ABB RAPID module: Robtargets.mod

MODULE Robtargets

    !**************************************************************************
    !ROBTARGET DECLARATIONS
    !**************************************************************************
    ! HOME AND STARTING Positions.

    CONST jointtarget AbsHome:=[[0,0,0,0,90,-60],[0,9E+09,9E+09,9E+09,9E+09,9E+09]];
    CONST robtarget Home:=[[351.01,0.00,709.09],[1.0026E-05,-3.87097E-05,1,4.46769E-06],[0,0,-1,0],[9E+09,9E+09,9E+09,9E+09,9E+09,9E+09]];
    CONST robtarget AboveStartAPosition:=[[68.84,70.35,87.16],[0.128377,0.734299,0.632585,-0.210145],[-1,-1,-1,0],[9E+09,9E+09,9E+09,9E+09,9E+09,9E+09]];
    CONST robtarget StartPosition:=[[68.84,70.35,87.16],[0.128377,0.734299,0.632585,-0.210145],[-1,-1,-1,0],[9E+09,9E+09,9E+09,9E+09,9E+09,9E+09]];
    CONST robtarget DicePickupPos:=[[-9.63,16.11,24.81],[0.0168056,0.706657,0.706736,-0.0296041],[-1,0,-2,0],[9E+09,9E+09,9E+09,9E+09,9E+09,9E+09]];
    CONST robtarget DiceThrowPos:=[[77.33,10.92,132.18],[0.0426025,0.942934,-0.0615583,-0.324456],[-2,0,-2,0],[9E+09,9E+09,9E+09,9E+09,9E+09,9E+09]];
    CONST robtarget DiceAbovePickPos:=[[-9.63,16.10,87.18],[0.0167928,0.706652,0.706742,-0.0296007],[-1,0,-2,0],[9E+09,9E+09,9E+09,9E+09,9E+09,9E+09]];

    CONST robtarget WinnerPos:=[[200.71,534.63,135.22],[0.00124171,-0.715438,-0.698667,-0.00340603],[0,0,0,0],[9E+09,9E+09,9E+09,9E+09,9E+09,9E+09]];
    CONST robtarget WinnerAbovePos:=[[200.71,534.63,260],[0.00124171,-0.715438,-0.698667,-0.00340603],[0,0,0,0],[9E+09,9E+09,9E+09,9E+09,9E+09,9E+09]];


    CONST robtarget Player1StartPos:=[[-39.27,392.54,23.61],[0.00279119,-0.701491,-0.712559,-0.0127358],[-1,-1,-1,0],[9E+09,9E+09,9E+09,9E+09,9E+09,9E+09]];
    CONST robtarget AbovePlayer1StartPos:=[[-39.27,392.54,200],[0.00279119,-0.701491,-0.712559,-0.0127358],[-1,-1,-1,0],[9E+09,9E+09,9E+09,9E+09,9E+09,9E+09]];
    CONST robtarget Player2StartPos:=[[-40.43,297.08,24.03],[0.00278384,-0.701482,-0.712569,-0.0126879],[-1,-1,-1,0],[9E+09,9E+09,9E+09,9E+09,9E+09,9E+09]];
    CONST robtarget AbovePlayer2StartPos:=[[-40.43,297.08,200],[0.00278384,-0.701482,-0.712569,-0.0126879],[-1,-1,-1,0],[9E+09,9E+09,9E+09,9E+09,9E+09,9E+09]];

    CONST robtarget Position00:=[[63.18,74.54,88.95],[0.138777,0.819807,0.520878,-0.193242],[-1,-1,0,0],[9E+09,9E+09,9E+09,9E+09,9E+09,9E+09]];
    CONST robtarget AbovePosition00:=[[63.18,74.54,200],[0.138777,0.819807,0.520878,-0.193242],[-1,-1,0,0],[9E+09,9E+09,9E+09,9E+09,9E+09,9E+09]];

    !1 TO 9
    CONST robtarget Position1:=[[118.73,66.16,87.22],[0.138793,0.819813,0.520859,-0.193257],[-1,-1,0,0],[9E+09,9E+09,9E+09,9E+09,9E+09,9E+09]];
    CONST robtarget AbovePosition1:=[[118.73,66.16,200],[0.138793,0.819813,0.520859,-0.193257],[-1,-1,0,0],[9E+09,9E+09,9E+09,9E+09,9E+09,9E+09]];

    CONST robtarget Position2:=[[177.20,64.51,84.69],[0.118125,0.704224,0.692906,-0.0999847],[-1,0,-1,0],[9E+09,9E+09,9E+09,9E+09,9E+09,9E+09]];
    CONST robtarget AbovePosition2:=[[177.20,64.51,200],[0.118125,0.704224,0.692906,-0.0999847],[-1,0,-1,0],[9E+09,9E+09,9E+09,9E+09,9E+09,9E+09]];

    CONST robtarget Position3:=[[231.06,64.54,84.66],[0.118102,0.704224,0.692915,-0.0999518],[-1,0,-1,0],[9E+09,9E+09,9E+09,9E+09,9E+09,9E+09]];
    CONST robtarget AbovePosition3:=[[231.06,64.54,200],[0.118102,0.704224,0.692915,-0.0999518],[-1,0,-1,0],[9E+09,9E+09,9E+09,9E+09,9E+09,9E+09]];

    CONST robtarget Position4:=[[283.24,64.54,84.66],[0.118095,0.704232,0.692908,-0.0999451],[0,0,-1,0],[9E+09,9E+09,9E+09,9E+09,9E+09,9E+09]];
    CONST robtarget AbovePosition4:=[[283.24,64.54,200],[0.118095,0.704232,0.692908,-0.0999451],[0,0,-1,0],[9E+09,9E+09,9E+09,9E+09,9E+09,9E+09]];

    CONST robtarget Position5:=[[336.21,64.54,84.66],[0.118088,0.704236,0.692906,-0.0999428],[0,-1,0,0],[9E+09,9E+09,9E+09,9E+09,9E+09,9E+09]];
    CONST robtarget AbovePosition5:=[[336.21,64.54,200],[0.118088,0.704236,0.692906,-0.0999428],[0,-1,0,0],[9E+09,9E+09,9E+09,9E+09,9E+09,9E+09]];

    CONST robtarget Position6:=[[388.67,64.54,84.66],[0.118113,0.704241,0.692895,-0.0999498],[0,-1,0,0],[9E+09,9E+09,9E+09,9E+09,9E+09,9E+09]];
    CONST robtarget AbovePosition6:=[[388.67,64.54,200],[0.118113,0.704241,0.692895,-0.0999498],[0,-1,0,0],[9E+09,9E+09,9E+09,9E+09,9E+09,9E+09]];

    CONST robtarget Position7:=[[439.75,64.55,84.60],[0.118098,0.704233,0.692908,-0.0999314],[0,-1,0,0],[9E+09,9E+09,9E+09,9E+09,9E+09,9E+09]];
    CONST robtarget AbovePosition7:=[[439.75,64.55,200],[0.118098,0.704233,0.692908,-0.0999314],[0,-1,0,0],[9E+09,9E+09,9E+09,9E+09,9E+09,9E+09]];

    CONST robtarget Position8:=[[491.75,69.67,84.56],[0.118087,0.704245,0.692902,-0.0999056],[0,-1,0,0],[9E+09,9E+09,9E+09,9E+09,9E+09,9E+09]];
    CONST robtarget AbovePosition8:=[[491.75,69.67,200],[0.118087,0.704245,0.692902,-0.0999056],[0,-1,0,0],[9E+09,9E+09,9E+09,9E+09,9E+09,9E+09]];

    CONST robtarget Position9:=[[510.49,108.79,84.55],[0.118067,0.70425,0.692902,-0.0998953],[0,-1,0,0],[9E+09,9E+09,9E+09,9E+09,9E+09,9E+09]];
    CONST robtarget AbovePosition9:=[[510.49,108.79,200],[0.118067,0.70425,0.692902,-0.0998953],[0,-1,0,0],[9E+09,9E+09,9E+09,9E+09,9E+09,9E+09]];

    CONST robtarget Position10:=[[476.96,151.88,84.56],[0.118067,0.704252,0.6929,-0.0998956],[0,-1,0,0],[9E+09,9E+09,9E+09,9E+09,9E+09,9E+09]];
    CONST robtarget AbovePosition10:=[[476.96,151.88,200],[0.118067,0.704252,0.6929,-0.0998956],[0,-1,0,0],[9E+09,9E+09,9E+09,9E+09,9E+09,9E+09]];


    !11 TO 20

    CONST robtarget Position11:=[[423.95,153.84,84.54],[0.118026,0.704242,0.69292,-0.0998776],[0,-1,0,0],[9E+09,9E+09,9E+09,9E+09,9E+09,9E+09]];
    CONST robtarget AbovePosition11:=[[423.95,153.84,200],[0.118026,0.704242,0.69292,-0.0998776],[0,-1,0,0],[9E+09,9E+09,9E+09,9E+09,9E+09,9E+09]];

    CONST robtarget Position12:=[[370.80,153.84,84.54],[0.118025,0.704242,0.692921,-0.0998746],[0,-1,0,0],[9E+09,9E+09,9E+09,9E+09,9E+09,9E+09]];
    CONST robtarget AbovePosition12:=[[370.80,153.84,200],[0.118025,0.704242,0.692921,-0.0998746],[0,-1,0,0],[9E+09,9E+09,9E+09,9E+09,9E+09,9E+09]];

    CONST robtarget Position13:=[[316.56,153.85,84.54],[0.118018,0.704245,0.692919,-0.0998685],[0,0,0,0],[9E+09,9E+09,9E+09,9E+09,9E+09,9E+09]];
    CONST robtarget AbovePosition13:=[[316.56,153.85,200],[0.118018,0.704245,0.692919,-0.0998685],[0,0,0,0],[9E+09,9E+09,9E+09,9E+09,9E+09,9E+09]];

    CONST robtarget Position14:=[[263.55,153.85,84.54],[0.118015,0.704243,0.692922,-0.0998641],[-1,0,-1,0],[9E+09,9E+09,9E+09,9E+09,9E+09,9E+09]];
    CONST robtarget AbovePosition14:=[[263.55,153.85,200],[0.118015,0.704243,0.692922,-0.0998641],[-1,0,-1,0],[9E+09,9E+09,9E+09,9E+09,9E+09,9E+09]];

    CONST robtarget Position15:=[[211.29,153.83,84.55],[0.118027,0.704235,0.692925,-0.0998929],[-1,0,-1,0],[9E+09,9E+09,9E+09,9E+09,9E+09,9E+09]];
    CONST robtarget AbovePosition15:=[[211.29,153.83,200],[0.118027,0.704235,0.692925,-0.0998929],[-1,0,-1,0],[9E+09,9E+09,9E+09,9E+09,9E+09,9E+09]];

    CONST robtarget Position16:=[[156.95,153.83,84.55],[0.118029,0.70423,0.692928,-0.0999031],[-1,0,-1,0],[9E+09,9E+09,9E+09,9E+09,9E+09,9E+09]];
    CONST robtarget AbovePosition16:=[[156.95,153.83,200],[0.118029,0.70423,0.692928,-0.0999031],[-1,0,-1,0],[9E+09,9E+09,9E+09,9E+09,9E+09,9E+09]];

    CONST robtarget Position17:=[[106.54,161.05,84.55],[0.118023,0.704218,0.69294,-0.0999059],[-1,0,-1,0],[9E+09,9E+09,9E+09,9E+09,9E+09,9E+09]];
    CONST robtarget AbovePosition17:=[[106.54,161.05,200],[0.118023,0.704218,0.69294,-0.0999059],[-1,0,-1,0],[9E+09,9E+09,9E+09,9E+09,9E+09,9E+09]];

    CONST robtarget Position18:=[[72.88,199.41,84.55],[0.118015,0.704204,0.692958,-0.0998897],[-1,0,-1,0],[9E+09,9E+09,9E+09,9E+09,9E+09,9E+09]];
    CONST robtarget AbovePosition18:=[[72.88,199.41,200],[0.118015,0.704204,0.692958,-0.0998897],[-1,0,-1,0],[9E+09,9E+09,9E+09,9E+09,9E+09,9E+09]];

    CONST robtarget Position19:=[[90.15,247.20,83.27],[0.00101801,-0.715468,-0.698638,-0.00318642],[-1,0,-1,0],[9E+09,9E+09,9E+09,9E+09,9E+09,9E+09]];
    CONST robtarget AbovePosition19:=[[90.15,247.20,200],[0.00101801,-0.715468,-0.698638,-0.00318642],[-1,0,-1,0],[9E+09,9E+09,9E+09,9E+09,9E+09,9E+09]];

    CONST robtarget Position20:=[[144.64,258.44,83.28],[0.00102727,-0.715462,-0.698643,-0.00319756],[-1,0,-1,0],[9E+09,9E+09,9E+09,9E+09,9E+09,9E+09]];
    CONST robtarget AbovePosition20:=[[144.64,258.44,200],[0.00102727,-0.715462,-0.698643,-0.00319756],[-1,0,-1,0],[9E+09,9E+09,9E+09,9E+09,9E+09,9E+09]];


    !21 TO 30

    CONST robtarget Position21:=[[197.53,258.45,83.28],[0.00104167,-0.715455,-0.69865,-0.00321534],[-1,0,-1,0],[9E+09,9E+09,9E+09,9E+09,9E+09,9E+09]];
    CONST robtarget AbovePosition21:=[[197.53,258.45,200],[0.00104167,-0.715455,-0.69865,-0.00321534],[-1,0,-1,0],[9E+09,9E+09,9E+09,9E+09,9E+09,9E+09]];

    CONST robtarget Position22:=[[251.56,258.46,83.29],[0.00104929,-0.715452,-0.698653,-0.00322303],[-1,0,-1,0],[9E+09,9E+09,9E+09,9E+09,9E+09,9E+09]];
    CONST robtarget AbovePosition22:=[[251.56,258.46,200],[0.00104929,-0.715452,-0.698653,-0.00322303],[-1,0,-1,0],[9E+09,9E+09,9E+09,9E+09,9E+09,9E+09]];

    CONST robtarget Position23:=[[304.12,258.46,83.28],[0.00104724,-0.715454,-0.698652,-0.00322172],[0,0,0,0],[9E+09,9E+09,9E+09,9E+09,9E+09,9E+09]];
    CONST robtarget AbovePosition23:=[[304.12,258.46,200],[0.00104724,-0.715454,-0.698652,-0.00322172],[0,0,0,0],[9E+09,9E+09,9E+09,9E+09,9E+09,9E+09]];

    CONST robtarget Position24:=[[355.55,258.45,83.28],[0.00102149,-0.715468,-0.698638,-0.00320467],[0,0,0,0],[9E+09,9E+09,9E+09,9E+09,9E+09,9E+09]];
    CONST robtarget AbovePosition24:=[[355.55,258.45,200],[0.00102149,-0.715468,-0.698638,-0.00320467],[0,0,0,0],[9E+09,9E+09,9E+09,9E+09,9E+09,9E+09]];

    CONST robtarget Position25:=[[409.67,258.45,83.28],[0.00101934,-0.715458,-0.698648,-0.0032026],[0,0,0,0],[9E+09,9E+09,9E+09,9E+09,9E+09,9E+09]];
    CONST robtarget AbovePosition25:=[[409.67,258.45,200],[0.00101934,-0.715458,-0.698648,-0.0032026],[0,0,0,0],[9E+09,9E+09,9E+09,9E+09,9E+09,9E+09]];

    CONST robtarget Position26:=[[464.38,260.32,83.27],[0.00103049,-0.715445,-0.698661,-0.00320834],[0,0,0,0],[9E+09,9E+09,9E+09,9E+09,9E+09,9E+09]];
    CONST robtarget AbovePosition26:=[[464.38,260.32,200],[0.00103049,-0.715445,-0.698661,-0.00320834],[0,0,0,0],[9E+09,9E+09,9E+09,9E+09,9E+09,9E+09]];

    CONST robtarget Position27:=[[494.41,301.60,83.28],[0.00104603,-0.715438,-0.698668,-0.00321548],[0,0,0,0],[9E+09,9E+09,9E+09,9E+09,9E+09,9E+09]];
    CONST robtarget AbovePosition27:=[[494.41,301.60,200],[0.00104603,-0.715438,-0.698668,-0.00321548],[0,0,0,0],[9E+09,9E+09,9E+09,9E+09,9E+09,9E+09]];

    CONST robtarget Position28:=[[481.35,349.43,83.26],[0.00107789,-0.715427,-0.698679,-0.00321957],[0,0,0,0],[9E+09,9E+09,9E+09,9E+09,9E+09,9E+09]];
    CONST robtarget AbovePosition28:=[[481.35,349.43,200],[0.00107789,-0.715427,-0.698679,-0.00321957],[0,0,0,0],[9E+09,9E+09,9E+09,9E+09,9E+09,9E+09]];

    CONST robtarget Position29:=[[428.33,351.84,83.26],[0.00109179,-0.715424,-0.698682,-0.00322696],[0,0,0,0],[9E+09,9E+09,9E+09,9E+09,9E+09,9E+09]];
    CONST robtarget AbovePosition29:=[[428.33,351.84,200],[0.00109179,-0.715424,-0.698682,-0.00322696],[0,0,0,0],[9E+09,9E+09,9E+09,9E+09,9E+09,9E+09]];

    CONST robtarget Position30:=[[375.36,351.85,83.26],[0.00110089,-0.715426,-0.69868,-0.00323293],[0,0,0,0],[9E+09,9E+09,9E+09,9E+09,9E+09,9E+09]];
    CONST robtarget AbovePosition30:=[[375.36,351.85,200],[0.00110089,-0.715426,-0.69868,-0.00323293],[0,0,0,0],[9E+09,9E+09,9E+09,9E+09,9E+09,9E+09]];


    !31 TO 40
    CONST robtarget Position31:=[[322.93,352.08,83.25],[0.00115336,-0.715442,-0.698663,-0.00327321],[0,-1,0,0],[9E+09,9E+09,9E+09,9E+09,9E+09,9E+09]];
    CONST robtarget AbovePosition31:=[[322.93,352.08,200],[0.00115336,-0.715442,-0.698663,-0.00327321],[0,-1,0,0],[9E+09,9E+09,9E+09,9E+09,9E+09,9E+09]];

    CONST robtarget Position32:=[[269.71,352.09,83.24],[0.00116463,-0.715448,-0.698657,-0.00328896],[-1,-1,-1,0],[9E+09,9E+09,9E+09,9E+09,9E+09,9E+09]];
    CONST robtarget AbovePosition32:=[[269.71,352.09,200],[0.00116463,-0.715448,-0.698657,-0.00328896],[-1,-1,-1,0],[9E+09,9E+09,9E+09,9E+09,9E+09,9E+09]];

    CONST robtarget Position33:=[[218.15,352.10,83.24],[0.00116707,-0.71544,-0.698665,-0.00328863],[-1,-1,-1,0],[9E+09,9E+09,9E+09,9E+09,9E+09,9E+09]];
    CONST robtarget AbovePosition33:=[[218.15,352.10,200],[0.00116707,-0.71544,-0.698665,-0.00328863],[-1,-1,-1,0],[9E+09,9E+09,9E+09,9E+09,9E+09,9E+09]];

    CONST robtarget Position34:=[[164.48,352.12,83.23],[0.00117983,-0.715427,-0.698678,-0.00331468],[-1,-1,-1,0],[9E+09,9E+09,9E+09,9E+09,9E+09,9E+09]];
    CONST robtarget AbovePosition34:=[[164.48,352.12,200],[0.00117983,-0.715427,-0.698678,-0.00331468],[-1,-1,-1,0],[9E+09,9E+09,9E+09,9E+09,9E+09,9E+09]];

    CONST robtarget Position35:=[[110.09,358.92,83.22],[0.00119315,-0.715427,-0.698679,-0.00334963],[-1,-1,-1,0],[9E+09,9E+09,9E+09,9E+09,9E+09,9E+09]];
    CONST robtarget AbovePosition35:=[[110.09,358.92,200],[0.00119315,-0.715427,-0.698679,-0.00334963],[-1,-1,-1,0],[9E+09,9E+09,9E+09,9E+09,9E+09,9E+09]];

    CONST robtarget Position36:=[[60.69,378.82,83.22],[0.00119013,-0.715425,-0.698681,-0.00333409],[-1,-1,-1,0],[9E+09,9E+09,9E+09,9E+09,9E+09,9E+09]];
    CONST robtarget AbovePosition36:=[[60.69,378.82,200],[0.00119013,-0.715425,-0.698681,-0.00333409],[-1,-1,-1,0],[9E+09,9E+09,9E+09,9E+09,9E+09,9E+09]];

    CONST robtarget Position37:=[[48.55,422.87,83.23],[0.00119175,-0.71543,-0.698675,-0.00333562],[-1,-1,-1,0],[9E+09,9E+09,9E+09,9E+09,9E+09,9E+09]];
    CONST robtarget AbovePosition37:=[[48.55,422.87,200],[0.00119175,-0.71543,-0.698675,-0.00333562],[-1,-1,-1,0],[9E+09,9E+09,9E+09,9E+09,9E+09,9E+09]];

    CONST robtarget Position38:=[[85.32,456.96,83.23],[0.00119527,-0.715427,-0.698679,-0.00335135],[-1,-1,-1,0],[9E+09,9E+09,9E+09,9E+09,9E+09,9E+09]];
    CONST robtarget AbovePosition38:=[[85.32,456.96,200],[0.00119527,-0.715427,-0.698679,-0.00335135],[-1,-1,-1,0],[9E+09,9E+09,9E+09,9E+09,9E+09,9E+09]];

    CONST robtarget Position39:=[[138.35,457.61,83.23],[0.00120429,-0.715433,-0.698672,-0.00338569],[-1,-1,-1,0],[9E+09,9E+09,9E+09,9E+09,9E+09,9E+09]];
    CONST robtarget AbovePosition39:=[[138.35,457.61,200],[0.00120429,-0.715433,-0.698672,-0.00338569],[-1,-1,-1,0],[9E+09,9E+09,9E+09,9E+09,9E+09,9E+09]];

    CONST robtarget Position40:=[[191.56,457.62,83.23],[0.00121366,-0.715427,-0.698678,-0.00340316],[-1,-1,-1,0],[9E+09,9E+09,9E+09,9E+09,9E+09,9E+09]];
    CONST robtarget AbovePosition40:=[[191.56,457.62,200],[0.00121366,-0.715427,-0.698678,-0.00340316],[-1,-1,-1,0],[9E+09,9E+09,9E+09,9E+09,9E+09,9E+09]];


    !41 TO 50
    CONST robtarget Position41:=[[245.02,457.62,83.23],[0.00121799,-0.715424,-0.698681,-0.00341009],[-1,-1,-1,0],[9E+09,9E+09,9E+09,9E+09,9E+09,9E+09]];
    CONST robtarget AbovePosition41:=[[245.02,457.62,200],[0.00121799,-0.715424,-0.698681,-0.00341009],[-1,-1,-1,0],[9E+09,9E+09,9E+09,9E+09,9E+09,9E+09]];

    CONST robtarget Position42:=[[297.02,457.62,83.22],[0.00121059,-0.715423,-0.698683,-0.00340594],[0,0,0,0],[9E+09,9E+09,9E+09,9E+09,9E+09,9E+09]];
    CONST robtarget AbovePosition42:=[[297.02,457.62,200],[0.00121059,-0.715423,-0.698683,-0.00340594],[0,0,0,0],[9E+09,9E+09,9E+09,9E+09,9E+09,9E+09]];

    CONST robtarget Position43:=[[350.67,457.62,83.22],[0.00120303,-0.715424,-0.698681,-0.00340147],[0,0,0,0],[9E+09,9E+09,9E+09,9E+09,9E+09,9E+09]];
    CONST robtarget AbovePosition43:=[[350.67,457.62,200],[0.00120303,-0.715424,-0.698681,-0.00340147],[0,0,0,0],[9E+09,9E+09,9E+09,9E+09,9E+09,9E+09]];

    CONST robtarget Position44:=[[405.00,457.61,83.22],[0.00118815,-0.71543,-0.698675,-0.0033961],[0,0,0,0],[9E+09,9E+09,9E+09,9E+09,9E+09,9E+09]];
    CONST robtarget AbovePosition44:=[[405.00,457.61,200],[0.00118815,-0.71543,-0.698675,-0.0033961],[0,0,0,0],[9E+09,9E+09,9E+09,9E+09,9E+09,9E+09]];

    CONST robtarget Position45:=[[455.85,457.60,83.22],[0.00114772,-0.715425,-0.69868,-0.00338543],[0,0,0,0],[9E+09,9E+09,9E+09,9E+09,9E+09,9E+09]];
    CONST robtarget AbovePosition45:=[[455.85,457.60,200],[0.00114772,-0.715425,-0.69868,-0.00338543],[0,0,0,0],[9E+09,9E+09,9E+09,9E+09,9E+09,9E+09]];

    CONST robtarget Position46:=[[498.76,483.63,83.22],[0.0011547,-0.715421,-0.698685,-0.0033882],[0,0,0,0],[9E+09,9E+09,9E+09,9E+09,9E+09,9E+09]];
    CONST robtarget AbovePosition46:=[[498.76,483.63,200],[0.0011547,-0.715421,-0.698685,-0.0033882],[0,0,0,0],[9E+09,9E+09,9E+09,9E+09,9E+09,9E+09]];

    CONST robtarget Position47:=[[492.42,526.12,83.22],[0.0011983,-0.715428,-0.698677,-0.00339119],[0,0,0,0],[9E+09,9E+09,9E+09,9E+09,9E+09,9E+09]];
    CONST robtarget AbovePosition47:=[[492.42,526.12,200],[0.0011983,-0.715428,-0.698677,-0.00339119],[0,0,0,0],[9E+09,9E+09,9E+09,9E+09,9E+09,9E+09]];

    CONST robtarget Position48:=[[442.47,534.62,83.22],[0.00121609,-0.715427,-0.698679,-0.00339529],[0,0,0,0],[9E+09,9E+09,9E+09,9E+09,9E+09,9E+09]];
    CONST robtarget AbovePosition48:=[[442.47,534.62,200],[0.00121609,-0.715427,-0.698679,-0.00339529],[0,0,0,0],[9E+09,9E+09,9E+09,9E+09,9E+09,9E+09]];

    CONST robtarget Position49:=[[388.24,534.63,83.22],[0.00123911,-0.71543,-0.698675,-0.00340311],[0,0,0,0],[9E+09,9E+09,9E+09,9E+09,9E+09,9E+09]];
    CONST robtarget AbovePosition49:=[[388.24,534.63,200],[0.00123911,-0.71543,-0.698675,-0.00340311],[0,0,0,0],[9E+09,9E+09,9E+09,9E+09,9E+09,9E+09]];

    CONST robtarget Position50:=[[332.71,534.63,83.22],[0.00124171,-0.715438,-0.698667,-0.00340603],[0,0,0,0],[9E+09,9E+09,9E+09,9E+09,9E+09,9E+09]];
    CONST robtarget AbovePosition50:=[[332.71,534.63,200],[0.00124171,-0.715438,-0.698667,-0.00340603],[0,0,0,0],[9E+09,9E+09,9E+09,9E+09,9E+09,9E+09]];


ENDMODULE
